// TIA Portal V20 export
DATA_BLOCK "SP508"   // DB324
// stored: MemoryReserve 100
   VAR
      "STACK-1 LIGHT CURTAIN OSSD 1" : Bool;
      "STACK-2 LIGHT CURTAIN OSSD 1" : Bool;
      "QR MARKING SHUTTER STATUS OUTPUT" : Bool;
      SPARE : Bool;
      "STACK-1 LIGHT CURTAIN OSSD 2" : Bool;
      "STACK-2 LIGHT CURTAIN OSSD 2" : Bool;
      SPARE_1 : Bool;
      SPARE_2 : Bool;
   END_VAR
BEGIN
END_DATA_BLOCK
